FUNCTION_BLOCK Persona
VAR_INPUT
END_VAR
VAR_OUTPUT
END_VAR
VAR
END_VAR

METHOD Comer
VAR_INPUT
END_VAR
END_METHOD

PROPERTY DNI : string
GET
END_GET
SET
END_SET
END_PROPERTY

END_FUNCTION_BLOCK

(* stored: Version 1.1.0.1, ProductVersion 3.1.4024.12
   POU Persona: Id {fc0af6d2-8453-444f-9721-4c38416cb952}, SpecialFunc None
   Method Comer: Id {8413425c-7d60-4a3e-89cd-a9d7ae047cda}
   Property DNI: Id {0931ebe7-5f8c-4611-9176-55939a6bbd7e}
   Get Get: Id {d8c31910-e7d6-475f-80e8-87d93fcc7aa5}
   Set Set: Id {ca4913ba-26d6-45a8-aec5-5bd376795a7a} *)
